// Mitsubishi GX Works2 project: Pract01_Contactos   PLC: FX3U/FX3UC

PROGRAM MAIN
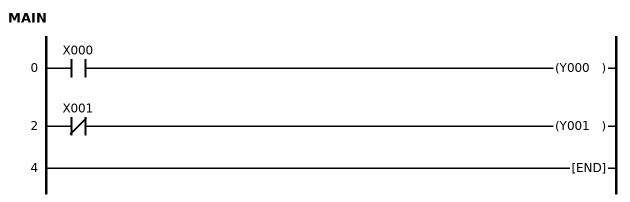
0     LD      X000
      OUT     Y000
2     LDI     X001
      OUT     Y001
4     END
END_PROGRAM
